// TIA Portal project "漳州" (V17)

(* hardware
DEVICE "S7-1200 station_1"  S7-1200 Station
   slot 0: "Rack_0"  S7-1200 Rack  Rack  V1.0
   slot 1: "PLC_1"  CPU 1215C AC/DC/Rly  6ES7 215-1BG40-0XB0  V4.3
   slot 2: "DI 16x24VDC/DQ 16xRelay_1"  SM 1223 DI16/DQ16 x relay  6ES7 223-1PL32-0XB0  V2.0
*)

// ===== PLC "PLC_1"  CPU 1215C AC/DC/Rly =====

VAR_GLOBAL   // PLC tag table "默认变量表"
   "启动" AT %I0.0 : Bool;
   "停止" AT %I0.1 : Bool;
   "变频器故障" AT %I0.5 : Bool;
   "有料检测" AT %I0.6 : Bool;
   "自动模式" AT %I0.3 : Bool;
   "分拣选择" AT %I0.2 : Bool;
   "变频器运行" AT %Q0.0 : Bool;
   "变频器速段" AT %Q0.1 : Bool;
   "1组正运行" AT %Q2.0 : Bool;
   "Tag_1" AT %Q3.0 : Bool;
   "2组正运行" AT %Q2.2 : Bool;
   "3组正运行" AT %Q2.4 : Bool;
   "4组正运行" AT %Q2.6 : Bool;
   "1组反转(1)" AT %Q2.1 : Bool;
   "2组反转(1)" AT %Q2.3 : Bool;
   "3组反转(1)" AT %Q2.5 : Bool;
   "4组反转(1)" AT %Q2.7 : Bool;
   "三基色绿色" AT %Q0.2 : Bool;
   "三基色红色" AT %Q0.4 : Bool;
   "蜂鸣器" AT %Q0.5 : Bool;
   "Tag_27" AT %Q3.1 : Bool;
   "Tag_28" AT %Q3.3 : Bool;
   "Tag_29" AT %Q3.5 : Bool;
   "Tag_30" AT %Q3.7 : Bool;
   "System_Byte" AT %MB1 : Byte;
   "FirstScan" AT %M1.0 : Bool;
   "DiagStatusUpdate" AT %M1.1 : Bool;
   "AlwaysTRUE" AT %M1.2 : Bool;
   "AlwaysFALSE" AT %M1.3 : Bool;
   "Clock_Byte" AT %MB0 : Byte;
   "Clock_10Hz" AT %M0.0 : Bool;
   "Clock_5Hz" AT %M0.1 : Bool;
   "Clock_2.5Hz" AT %M0.2 : Bool;
   "Clock_2Hz" AT %M0.3 : Bool;
   "Clock_1.25Hz" AT %M0.4 : Bool;
   "Clock_1Hz" AT %M0.5 : Bool;
   "Clock_0.625Hz" AT %M0.6 : Bool;
   "Clock_0.5Hz" AT %M0.7 : Bool;
   "系统启动" AT %M2.0 : Bool;
   "Tag_2" AT %M2.1 : Bool;
   "Tag_3" AT %MW100 : Word;
   "Tag_4" AT %M2.2 : Bool;
   "1组运转" AT %M3.0 : Bool;
   "1组正转" AT %M3.1 : Bool;
   "2组运转" AT %M3.2 : Bool;
   "2组正转" AT %M3.3 : Bool;
   "Tag_5" AT %M20.0 : Bool;
   "3组运转" AT %M3.4 : Bool;
   "3组正转" AT %M3.5 : Bool;
   "4组运转" AT %M3.6 : Bool;
   "4组正转" AT %M3.7 : Bool;
   "1组反运行" AT %M4.0 : Bool;
   "1组反转" AT %M4.1 : Bool;
   "2组反运转" AT %M4.2 : Bool;
   "2组反转" AT %M4.3 : Bool;
   "3组反运行" AT %M4.4 : Bool;
   "3组反转" AT %M4.5 : Bool;
   "4组反运行" AT %M4.6 : Bool;
   "4组反转" AT %M4.7 : Bool;
   "Tag_6" AT %M20.1 : Bool;
   "Tag_7" AT %M20.2 : Bool;
   "Tag_8" AT %M20.3 : Bool;
   "Tag_9" AT %MW200 : Int;
   "Tag_10" AT %MW201 : Int;
   "Tag_11" AT %MW202 : Int;
   "Tag_12" AT %MW203 : Int;
   "Tag_13" AT %MW204 : Int;
   "Tag_14" AT %MW205 : Int;
   "Tag_15" AT %MW206 : Int;
   "Tag_16" AT %MW300 : Int;
   "Tag_17" AT %MW302 : Int;
   "Tag_18" AT %MW304 : Int;
   "Tag_19" AT %MW306 : Int;
   "Tag_20" AT %M110.0 : Bool;
   "Tag_21" AT %MD200 : DWord;
   "Tag_22" AT %MD300 : DWord;
   "Tag_23" AT %MD204 : DWord;
   "Tag_24" AT %MD304 : DWord;
   "Tag_25" AT %M100.0 : Bool;
   "Tag_26" AT %M200.0 : Bool;
   "Tag_31" AT %M200.1 : Bool;
   "Tag_32" AT %M200.2 : Bool;
   "Tag_33" AT %M300.0 : Bool;
   "Tag_34" AT %M5.2 : Bool;
   "Tag_35" AT %M5.3 : Bool;
   "Tag_36" AT %M5.4 : Bool;
   "Tag_37" AT %M11.0 : Bool;
   "Tag_38" AT %M101.0 : Bool;
   "Tag_39" AT %M12.0 : Bool;
   "Tag_40" AT %M12.1 : Bool;
   "Tag_41" AT %M12.2 : Bool;
   "Tag_42" AT %M12.3 : Bool;
   "Tag_43" AT %M12.4 : Bool;
   "Tag_44" AT %M12.5 : Bool;
   "Tag_45" AT %M12.6 : Bool;
   "Tag_46" AT %MB10 : Byte;
   "5组正转" AT %M5.0 : Bool;
   "Tag_48" AT %M6.1 : Bool;
   "Tag_49" AT %M6.2 : Bool;
   "Tag_50" AT %M6.3 : Bool;
   "Tag_51" AT %M6.4 : Bool;
   "Tag_52" AT %M6.5 : Bool;
   "Tag_53" AT %M6.6 : Bool;
   "Tag_54" AT %M6.7 : Bool;
   "Tag_55" AT %M6.0 : Bool;
   "Tag_56" AT %M90.3 : Bool;
   "Tag_57" AT %M90.5 : Bool;
   "Tag_58" AT %M90.0 : Bool;
   "Tag_59" AT %M7.0 : Bool;
   "Tag_60" AT %M7.1 : Bool;
   "Tag_61" AT %M90.2 : Bool;
   "Tag_62" AT %M90.1 : Bool;
   "Tag_63" AT %M7.2 : Bool;
   "Tag_64" AT %M7.3 : Bool;
   "Tag_65" AT %M90.4 : Bool;
   "Tag_66" AT %M7.4 : Bool;
   "Tag_67" AT %M7.5 : Bool;
   "Tag_68" AT %M7.6 : Bool;
   "Tag_69" AT %M8.0 : Bool;
   "Tag_70" AT %M8.1 : Bool;
   "Tag_71" AT %M8.2 : Bool;
   "Tag_72" AT %M8.3 : Bool;
   "Tag_73" AT %M8.4 : Bool;
   "Tag_74" AT %M8.5 : Bool;
   "Tag_75" AT %M8.6 : Bool;
   "Tag_76" AT %M8.7 : Bool;
   "5组反转" AT %M5.1 : Bool;
   "Tag_78" AT %MW102 : Word;
   "Tag_79" AT %MB100 : Byte;
   "Tag_80" AT %M5.5 : Bool;
   "1-1口计时" AT %M10.0 : Bool;
   "1-2计时" AT %M10.1 : Bool;
   "Tag_82" AT %Q10.0 : Bool;
   "Tag_83" AT %M101.1 : Bool;
   "Tag_84" AT %M101.2 : Bool;
   "Tag_81" AT %Q10.1 : Bool;
   "Tag_85" AT %M101.3 : Bool;
   "Tag_86" AT %M10.2 : Bool;
   "Tag_87" AT %Q10.2 : Bool;
   "Tag_88" AT %M101.4 : Bool;
   "Tag_89" AT %M10.3 : Bool;
   "Tag_90" AT %M101.5 : Bool;
   "Tag_91" AT %M101.6 : Bool;
   "Tag_92" AT %M101.7 : Bool;
   "Tag_93" AT %MB101 : Byte;
   "Tag_94" AT %M100.1 : Bool;
   "Tag_95" AT %M100.2 : Bool;
   "Tag_96" AT %M100.3 : Bool;
   "Tag_97" AT %M100.4 : Bool;
   "Tag_98" AT %MB102 : Byte;
   "Tag_99" AT %MB103 : Byte;
   "Tag_100" AT %M103.1 : Bool;
   "Tag_101" AT %M102.2 : Bool;
   "Tag_102" AT %M102.3 : Bool;
   "Tag_103" AT %M102.4 : Bool;
   "Tag_104" AT %M103.2 : Bool;
   "Tag_105" AT %M103.3 : Bool;
   "Tag_106" AT %M103.4 : Bool;
   "Tag_107" AT %M102.1 : Bool;
   "Tag_108" AT %MB104 : Byte;
   "Tag_109" AT %MB105 : Byte;
   "Tag_110" AT %M105.1 : Bool;
   "Tag_111" AT %M105.2 : Bool;
   "Tag_112" AT %M105.3 : Bool;
   "Tag_113" AT %M105.4 : Bool;
   "Tag_114" AT %M104.1 : Bool;
   "Tag_115" AT %M104.2 : Bool;
   "Tag_116" AT %M104.3 : Bool;
   "Tag_117" AT %MB106 : Byte;
   "Tag_118" AT %MB107 : Byte;
   "Tag_119" AT %M107.1 : Bool;
   "Tag_120" AT %M107.2 : Bool;
   "Tag_121" AT %M107.3 : Bool;
   "Tag_122" AT %M107.4 : Bool;
   "Tag_123" AT %M106.1 : Bool;
   "Tag_124" AT %M106.2 : Bool;
   "Tag_125" AT %M106.3 : Bool;
   "Tag_126" AT %M106.4 : Bool;
   "Tag_127" AT %MB108 : Byte;
   "Tag_128" AT %MB109 : Byte;
   "Tag_129" AT %M109.1 : Bool;
   "Tag_130" AT %M109.2 : Bool;
   "Tag_131" AT %M109.3 : Bool;
   "Tag_132" AT %M109.4 : Bool;
   "Tag_133" AT %M109.5 : Bool;
   "Tag_134" AT %M108.1 : Bool;
   "Tag_135" AT %M108.2 : Bool;
   "Tag_136" AT %M108.3 : Bool;
   "Tag_137" AT %M108.4 : Bool;
   "Tag_138" AT %M108.5 : Bool;
END_VAR

TYPE "用户数据类型_1"
   STRUCT
      Q : Array[0..12] of Bool;
   END_STRUCT;
END_TYPE

DATA_BLOCK "1口_DB"   // DB1
{ S7_Optimized_Access := 'TRUE' }
VERSION : 0.1
// stored: InstanceOfName 1口
"1口"
BEGIN
END_DATA_BLOCK

DATA_BLOCK "2口_DB"   // DB2
{ S7_Optimized_Access := 'TRUE' }
VERSION : 0.1
// stored: InstanceOfName 2口
"2口"
BEGIN
END_DATA_BLOCK

DATA_BLOCK "3口_DB"   // DB3
{ S7_Optimized_Access := 'TRUE' }
VERSION : 0.1
// stored: InstanceOfName 3口
"3口"
BEGIN
END_DATA_BLOCK

DATA_BLOCK "4口_DB"   // DB4
{ S7_Optimized_Access := 'TRUE' }
VERSION : 0.1
// stored: InstanceOfName 4口
"4口"
BEGIN
END_DATA_BLOCK

DATA_BLOCK "数据块_1"   // DB5
{ S7_Optimized_Access := 'TRUE' }
VERSION : 0.1
   VAR
      箱号 : Int;
      分拣时间 : Time := T#1s;
      到达时间 : Time := T#10s;
      光电 : Bool;
      计数 : Bool;
      Q : Array[0..12] of Bool;
   END_VAR
BEGIN
END_DATA_BLOCK

DATA_BLOCK "5口_DB"   // DB6
{ S7_Optimized_Access := 'TRUE' }
VERSION : 0.1
// stored: InstanceOfName 5口
"5口"
BEGIN
END_DATA_BLOCK

FUNCTION_BLOCK "1口"   // FB1, LAD
{ S7_Optimized_Access := 'TRUE' }
VERSION : 0.1
   VAR_INPUT
      光电 : Bool;
      箱号 : Int;
   END_VAR
   VAR_OUTPUT
      Q : Array[0..12] of Bool;
   END_VAR
   VAR
      TON_TIME : Array[0..21] of TON_TIME;
      IEC_Timer : Array[0..11] of IEC_TIMER;
      "M" : Array[0..11] of Bool;
      M1 : Array[0..11] of Bool;
      光电上升沿 : Array[0..2] of Bool;
   END_VAR
   VAR_TEMP   // added for the SCL form of the ladder/FBD networks
      _w1 : Bool;
      _w2 : Bool;
      _w3 : Bool;
   END_VAR
BEGIN

REGION Network 1: 记录箱号
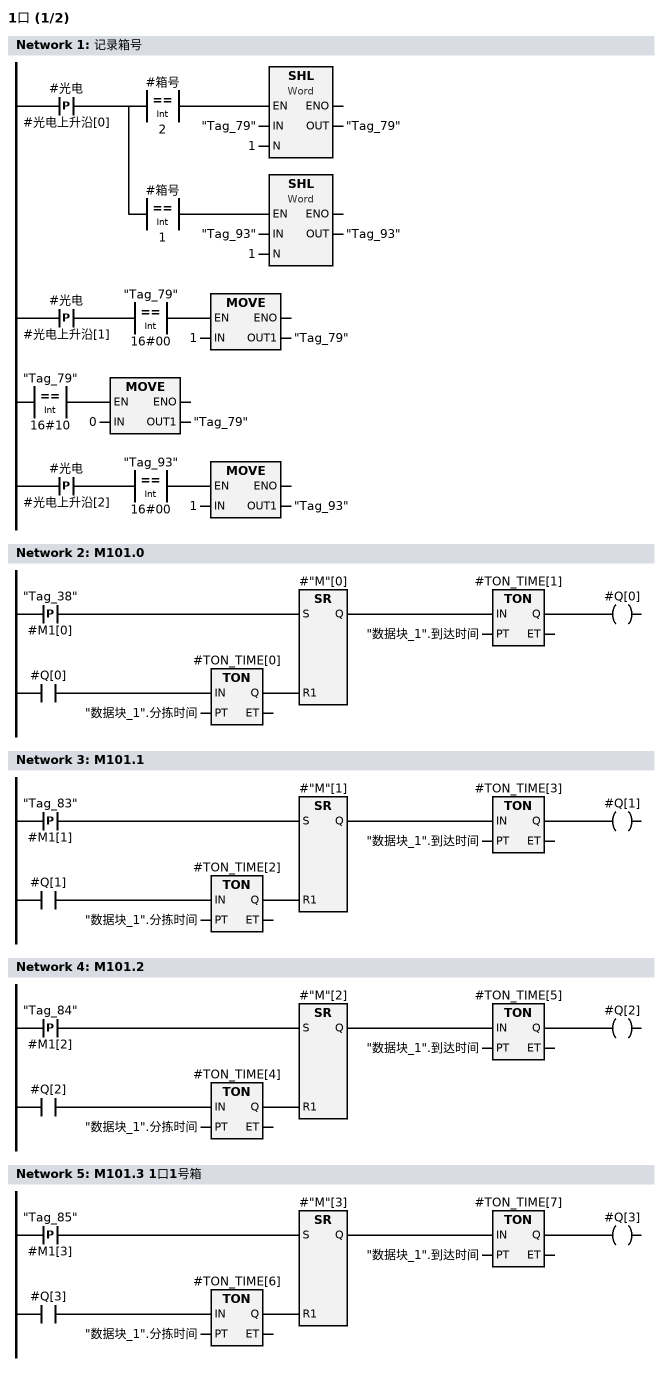
   RUNG wire#powerrail
      P_Contact(operand := #光电, bit := #光电上升沿[0])
      wire#w1
      { S7_Templates := "SrcType := Int" } EQ_Contact(in1 := #箱号, in2 := 2)
      { S7_Templates := "SrcType := Word" } Shl(in := "Tag_79", n := 1, out => "Tag_79")
   END_RUNG
   RUNG wire#w1
      { S7_Templates := "SrcType := Int" } EQ_Contact(in1 := #箱号, in2 := 1)
      { S7_Templates := "SrcType := Word" } Shl(in := "Tag_93", n := 1, out => "Tag_93")
   END_RUNG
   RUNG wire#powerrail
      P_Contact(operand := #光电, bit := #光电上升沿[1])
      { S7_Templates := "SrcType := Int" } EQ_Contact(in1 := "Tag_79", in2 := 16#00)
      Move(in := 1, out1 => "Tag_79")
   END_RUNG
   RUNG wire#powerrail
      { S7_Templates := "SrcType := Int" } EQ_Contact(in1 := "Tag_79", in2 := 16#10)
      Move(in := 0, out1 => "Tag_79")
   END_RUNG
   RUNG wire#powerrail
      P_Contact(operand := #光电, bit := #光电上升沿[2])
      { S7_Templates := "SrcType := Int" } EQ_Contact(in1 := "Tag_93", in2 := 16#00)
      Move(in := 1, out1 => "Tag_93")
   END_RUNG
   // the same network as SCL:
   #_w1 := #光电 AND NOT #光电上升沿[0];   // rising edge of #光电
   #光电上升沿[0] := #光电;
   IF #_w1 AND (#箱号 = 2) THEN "Tag_79" := SHL(IN := "Tag_79", N := 1); END_IF;
   IF #_w1 AND (#箱号 = 1) THEN "Tag_93" := SHL(IN := "Tag_93", N := 1); END_IF;
   #_w2 := #光电 AND NOT #光电上升沿[1];   // rising edge of #光电
   #光电上升沿[1] := #光电;
   IF #_w2 AND ("Tag_79" = 16#00) THEN "Tag_79" := 1; END_IF;
   IF "Tag_79" = 16#10 THEN "Tag_79" := 0; END_IF;
   #_w3 := #光电 AND NOT #光电上升沿[2];   // rising edge of #光电
   #光电上升沿[2] := #光电;
   IF #_w3 AND ("Tag_93" = 16#00) THEN "Tag_93" := 1; END_IF;
END_REGION

REGION Network 2: M101.0
   #_w1 := "Tag_38" AND NOT #M1[0];   // rising edge of "Tag_38"
   #M1[0] := "Tag_38";
   #TON_TIME[0].TON(IN := #Q[0], PT := "数据块_1".分拣时间);
   IF #_w1 THEN
       #"M"[0] := TRUE;   // SR flip-flop
   END_IF;
   IF #TON_TIME[0].Q THEN #"M"[0] := FALSE; END_IF;
   #TON_TIME[1].TON(IN := #"M"[0], PT := "数据块_1".到达时间);
   #Q[0] := #TON_TIME[1].Q;
END_REGION

REGION Network 3: M101.1
   #_w1 := "Tag_83" AND NOT #M1[1];   // rising edge of "Tag_83"
   #M1[1] := "Tag_83";
   #TON_TIME[2].TON(IN := #Q[1], PT := "数据块_1".分拣时间);
   IF #_w1 THEN
       #"M"[1] := TRUE;   // SR flip-flop
   END_IF;
   IF #TON_TIME[2].Q THEN #"M"[1] := FALSE; END_IF;
   #TON_TIME[3].TON(IN := #"M"[1], PT := "数据块_1".到达时间);
   #Q[1] := #TON_TIME[3].Q;
END_REGION

REGION Network 4: M101.2
   #_w1 := "Tag_84" AND NOT #M1[2];   // rising edge of "Tag_84"
   #M1[2] := "Tag_84";
   #TON_TIME[4].TON(IN := #Q[2], PT := "数据块_1".分拣时间);
   IF #_w1 THEN
       #"M"[2] := TRUE;   // SR flip-flop
   END_IF;
   IF #TON_TIME[4].Q THEN #"M"[2] := FALSE; END_IF;
   #TON_TIME[5].TON(IN := #"M"[2], PT := "数据块_1".到达时间);
   #Q[2] := #TON_TIME[5].Q;
END_REGION

REGION Network 5: M101.3 1口1号箱
   #_w1 := "Tag_85" AND NOT #M1[3];   // rising edge of "Tag_85"
   #M1[3] := "Tag_85";
   #TON_TIME[6].TON(IN := #Q[3], PT := "数据块_1".分拣时间);
   IF #_w1 THEN
       #"M"[3] := TRUE;   // SR flip-flop
   END_IF;
   IF #TON_TIME[6].Q THEN #"M"[3] := FALSE; END_IF;
   #TON_TIME[7].TON(IN := #"M"[3], PT := "数据块_1".到达时间);
   #Q[3] := #TON_TIME[7].Q;
END_REGION

REGION Network 6: M100.0 1口2号箱
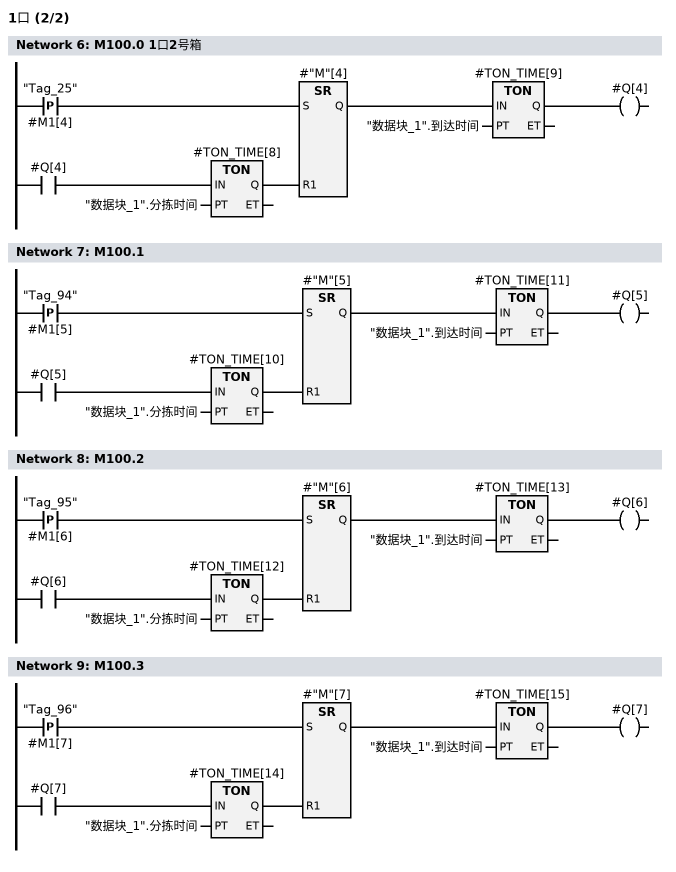
   #_w1 := "Tag_25" AND NOT #M1[4];   // rising edge of "Tag_25"
   #M1[4] := "Tag_25";
   #TON_TIME[8].TON(IN := #Q[4], PT := "数据块_1".分拣时间);
   IF #_w1 THEN
       #"M"[4] := TRUE;   // SR flip-flop
   END_IF;
   IF #TON_TIME[8].Q THEN #"M"[4] := FALSE; END_IF;
   #TON_TIME[9].TON(IN := #"M"[4], PT := "数据块_1".到达时间);
   #Q[4] := #TON_TIME[9].Q;
END_REGION

REGION Network 7: M100.1
   #_w1 := "Tag_94" AND NOT #M1[5];   // rising edge of "Tag_94"
   #M1[5] := "Tag_94";
   #TON_TIME[10].TON(IN := #Q[5], PT := "数据块_1".分拣时间);
   IF #_w1 THEN
       #"M"[5] := TRUE;   // SR flip-flop
   END_IF;
   IF #TON_TIME[10].Q THEN #"M"[5] := FALSE; END_IF;
   #TON_TIME[11].TON(IN := #"M"[5], PT := "数据块_1".到达时间);
   #Q[5] := #TON_TIME[11].Q;
END_REGION

REGION Network 8: M100.2
   #_w1 := "Tag_95" AND NOT #M1[6];   // rising edge of "Tag_95"
   #M1[6] := "Tag_95";
   #TON_TIME[12].TON(IN := #Q[6], PT := "数据块_1".分拣时间);
   IF #_w1 THEN
       #"M"[6] := TRUE;   // SR flip-flop
   END_IF;
   IF #TON_TIME[12].Q THEN #"M"[6] := FALSE; END_IF;
   #TON_TIME[13].TON(IN := #"M"[6], PT := "数据块_1".到达时间);
   #Q[6] := #TON_TIME[13].Q;
END_REGION

REGION Network 9: M100.3
   #_w1 := "Tag_96" AND NOT #M1[7];   // rising edge of "Tag_96"
   #M1[7] := "Tag_96";
   #TON_TIME[14].TON(IN := #Q[7], PT := "数据块_1".分拣时间);
   IF #_w1 THEN
       #"M"[7] := TRUE;   // SR flip-flop
   END_IF;
   IF #TON_TIME[14].Q THEN #"M"[7] := FALSE; END_IF;
   #TON_TIME[15].TON(IN := #"M"[7], PT := "数据块_1".到达时间);
   #Q[7] := #TON_TIME[15].Q;
END_REGION

REGION Network 10 (SCL)
   IF #Q[0] OR #Q[1] OR #Q[2] OR #Q[3] THEN
       "1组正转" := TRUE;
   ELSE
       "1组正转" := FALSE;
   END_IF;

   IF #Q[4] OR #Q[5] OR #Q[6] OR #Q[7] THEN
       "1组反转" := TRUE;
   ELSE
       "1组反转" := FALSE;
   END_IF;
END_REGION
END_FUNCTION_BLOCK

FUNCTION_BLOCK "2口"   // FB2, LAD
{ S7_Optimized_Access := 'TRUE' }
VERSION : 0.1
   VAR_INPUT
      光电 : Bool;
      箱号 : Int;
   END_VAR
   VAR_OUTPUT
      Q : Array[0..12] of Bool;
   END_VAR
   VAR
      TON_TIME : Array[0..21] of TON_TIME;
      IEC_Timer : Array[0..11] of IEC_TIMER;
      "M" : Array[0..11] of Bool;
      M1 : Array[0..11] of Bool;
      光电上升沿 : Bool;
   END_VAR
   VAR_TEMP   // added for the SCL form of the ladder/FBD networks
      _w1 : Bool;
      _w2 : Bool;
      _w3 : Bool;
   END_VAR
BEGIN

REGION Network 1: 记录箱号
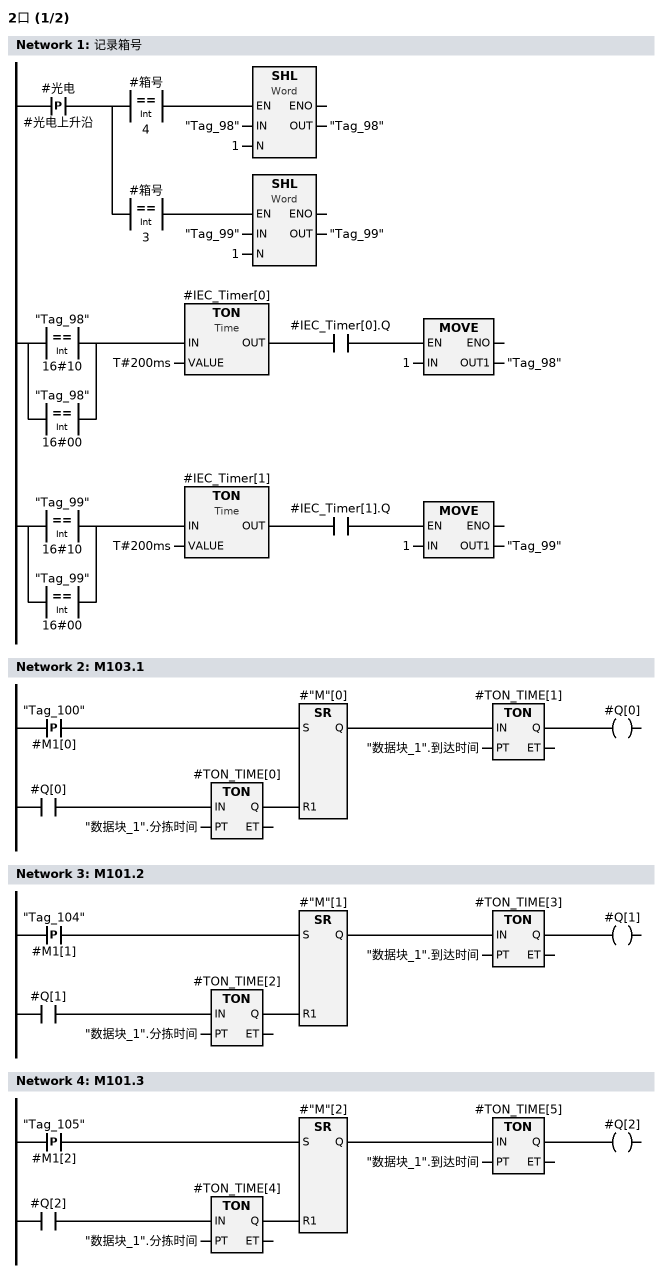
   #_w1 := #光电 AND NOT #光电上升沿;   // rising edge of #光电
   #光电上升沿 := #光电;
   IF #_w1 AND (#箱号 = 4) THEN "Tag_98" := SHL(IN := "Tag_98", N := 1); END_IF;
   IF #_w1 AND (#箱号 = 3) THEN "Tag_99" := SHL(IN := "Tag_99", N := 1); END_IF;
   #_w2 := ("Tag_98" = 16#10) OR ("Tag_98" = 16#00);
   #IEC_Timer[0].TON(IN := #_w2, PT := T#200ms);   // TON coil
   IF #_w2 AND #IEC_Timer[0].Q THEN "Tag_98" := 1; END_IF;
   #_w3 := ("Tag_99" = 16#10) OR ("Tag_99" = 16#00);
   #IEC_Timer[1].TON(IN := #_w3, PT := T#200ms);   // TON coil
   IF #_w3 AND #IEC_Timer[1].Q THEN "Tag_99" := 1; END_IF;
END_REGION

REGION Network 2: M103.1
   #_w1 := "Tag_100" AND NOT #M1[0];   // rising edge of "Tag_100"
   #M1[0] := "Tag_100";
   #TON_TIME[0].TON(IN := #Q[0], PT := "数据块_1".分拣时间);
   IF #_w1 THEN
       #"M"[0] := TRUE;   // SR flip-flop
   END_IF;
   IF #TON_TIME[0].Q THEN #"M"[0] := FALSE; END_IF;
   #TON_TIME[1].TON(IN := #"M"[0], PT := "数据块_1".到达时间);
   #Q[0] := #TON_TIME[1].Q;
END_REGION

REGION Network 3: M101.2
   #_w1 := "Tag_104" AND NOT #M1[1];   // rising edge of "Tag_104"
   #M1[1] := "Tag_104";
   #TON_TIME[2].TON(IN := #Q[1], PT := "数据块_1".分拣时间);
   IF #_w1 THEN
       #"M"[1] := TRUE;   // SR flip-flop
   END_IF;
   IF #TON_TIME[2].Q THEN #"M"[1] := FALSE; END_IF;
   #TON_TIME[3].TON(IN := #"M"[1], PT := "数据块_1".到达时间);
   #Q[1] := #TON_TIME[3].Q;
END_REGION

REGION Network 4: M101.3
   #_w1 := "Tag_105" AND NOT #M1[2];   // rising edge of "Tag_105"
   #M1[2] := "Tag_105";
   #TON_TIME[4].TON(IN := #Q[2], PT := "数据块_1".分拣时间);
   IF #_w1 THEN
       #"M"[2] := TRUE;   // SR flip-flop
   END_IF;
   IF #TON_TIME[4].Q THEN #"M"[2] := FALSE; END_IF;
   #TON_TIME[5].TON(IN := #"M"[2], PT := "数据块_1".到达时间);
   #Q[2] := #TON_TIME[5].Q;
END_REGION

REGION Network 5: M101.4 1口1号箱
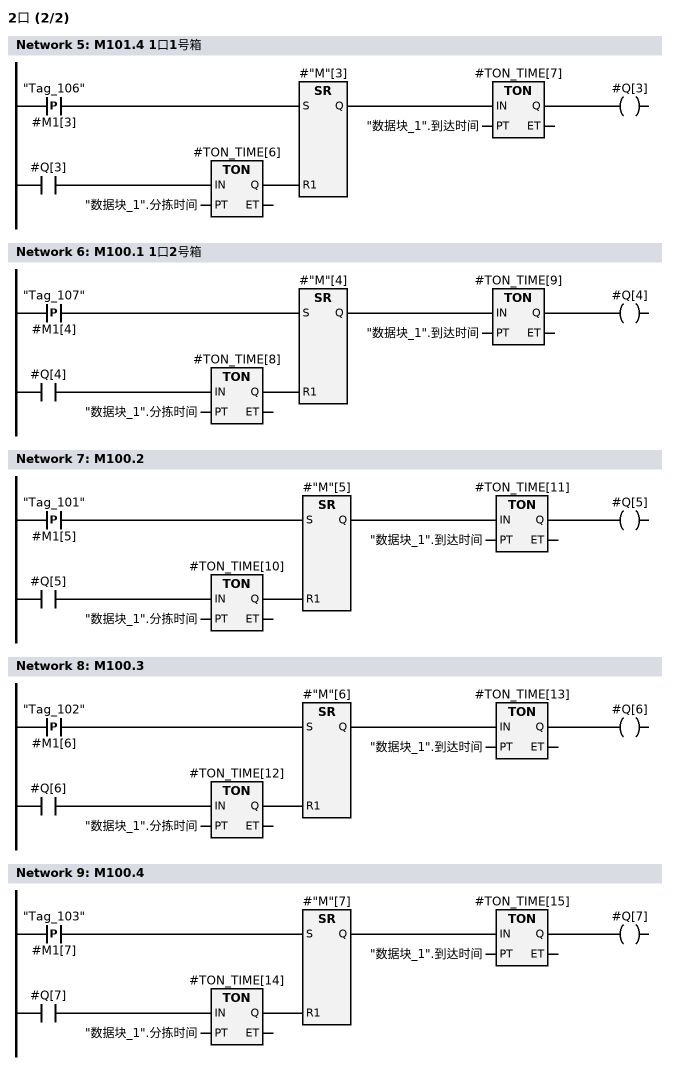
   #_w1 := "Tag_106" AND NOT #M1[3];   // rising edge of "Tag_106"
   #M1[3] := "Tag_106";
   #TON_TIME[6].TON(IN := #Q[3], PT := "数据块_1".分拣时间);
   IF #_w1 THEN
       #"M"[3] := TRUE;   // SR flip-flop
   END_IF;
   IF #TON_TIME[6].Q THEN #"M"[3] := FALSE; END_IF;
   #TON_TIME[7].TON(IN := #"M"[3], PT := "数据块_1".到达时间);
   #Q[3] := #TON_TIME[7].Q;
END_REGION

REGION Network 6: M100.1 1口2号箱
   #_w1 := "Tag_107" AND NOT #M1[4];   // rising edge of "Tag_107"
   #M1[4] := "Tag_107";
   #TON_TIME[8].TON(IN := #Q[4], PT := "数据块_1".分拣时间);
   IF #_w1 THEN
       #"M"[4] := TRUE;   // SR flip-flop
   END_IF;
   IF #TON_TIME[8].Q THEN #"M"[4] := FALSE; END_IF;
   #TON_TIME[9].TON(IN := #"M"[4], PT := "数据块_1".到达时间);
   #Q[4] := #TON_TIME[9].Q;
END_REGION

REGION Network 7: M100.2
   #_w1 := "Tag_101" AND NOT #M1[5];   // rising edge of "Tag_101"
   #M1[5] := "Tag_101";
   #TON_TIME[10].TON(IN := #Q[5], PT := "数据块_1".分拣时间);
   IF #_w1 THEN
       #"M"[5] := TRUE;   // SR flip-flop
   END_IF;
   IF #TON_TIME[10].Q THEN #"M"[5] := FALSE; END_IF;
   #TON_TIME[11].TON(IN := #"M"[5], PT := "数据块_1".到达时间);
   #Q[5] := #TON_TIME[11].Q;
END_REGION

REGION Network 8: M100.3
   #_w1 := "Tag_102" AND NOT #M1[6];   // rising edge of "Tag_102"
   #M1[6] := "Tag_102";
   #TON_TIME[12].TON(IN := #Q[6], PT := "数据块_1".分拣时间);
   IF #_w1 THEN
       #"M"[6] := TRUE;   // SR flip-flop
   END_IF;
   IF #TON_TIME[12].Q THEN #"M"[6] := FALSE; END_IF;
   #TON_TIME[13].TON(IN := #"M"[6], PT := "数据块_1".到达时间);
   #Q[6] := #TON_TIME[13].Q;
END_REGION

REGION Network 9: M100.4
   #_w1 := "Tag_103" AND NOT #M1[7];   // rising edge of "Tag_103"
   #M1[7] := "Tag_103";
   #TON_TIME[14].TON(IN := #Q[7], PT := "数据块_1".分拣时间);
   IF #_w1 THEN
       #"M"[7] := TRUE;   // SR flip-flop
   END_IF;
   IF #TON_TIME[14].Q THEN #"M"[7] := FALSE; END_IF;
   #TON_TIME[15].TON(IN := #"M"[7], PT := "数据块_1".到达时间);
   #Q[7] := #TON_TIME[15].Q;
END_REGION

REGION Network 10 (SCL)
   IF #Q[0] OR #Q[1] OR #Q[2] OR #Q[3] THEN
       "2组正转" := TRUE;
   ELSE
       "2组正转" := FALSE;
   END_IF;

   IF #Q[4] OR #Q[5] OR #Q[6] OR #Q[7] THEN
       "2组反转" := TRUE;
   ELSE
       "2组反转" := FALSE;
   END_IF;
END_REGION
END_FUNCTION_BLOCK

FUNCTION_BLOCK "3口"   // FB3, LAD
{ S7_Optimized_Access := 'TRUE' }
VERSION : 0.1
   VAR_INPUT
      光电 : Bool;
      箱号 : Int;
   END_VAR
   VAR_OUTPUT
      Q : Array[0..12] of Bool;
   END_VAR
   VAR
      TON_TIME : Array[0..21] of TON_TIME;
      IEC_Timer : Array[0..11] of IEC_TIMER;
      "M" : Array[0..11] of Bool;
      M1 : Array[0..11] of Bool;
      光电上升沿 : Bool;
   END_VAR
   VAR_TEMP   // added for the SCL form of the ladder/FBD networks
      _w1 : Bool;
      _w2 : Bool;
      _w3 : Bool;
   END_VAR
BEGIN

REGION Network 1: 记录箱号
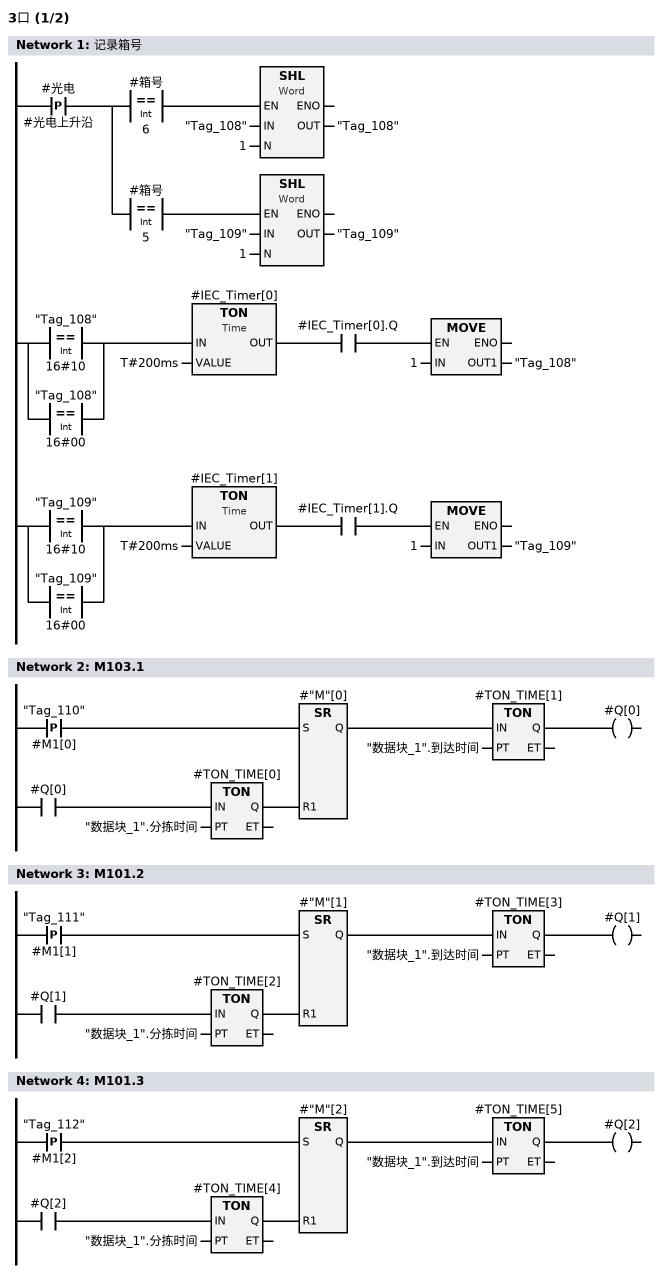
   #_w1 := #光电 AND NOT #光电上升沿;   // rising edge of #光电
   #光电上升沿 := #光电;
   IF #_w1 AND (#箱号 = 6) THEN "Tag_108" := SHL(IN := "Tag_108", N := 1); END_IF;
   IF #_w1 AND (#箱号 = 5) THEN "Tag_109" := SHL(IN := "Tag_109", N := 1); END_IF;
   #_w2 := ("Tag_108" = 16#10) OR ("Tag_108" = 16#00);
   #IEC_Timer[0].TON(IN := #_w2, PT := T#200ms);   // TON coil
   IF #_w2 AND #IEC_Timer[0].Q THEN "Tag_108" := 1; END_IF;
   #_w3 := ("Tag_109" = 16#10) OR ("Tag_109" = 16#00);
   #IEC_Timer[1].TON(IN := #_w3, PT := T#200ms);   // TON coil
   IF #_w3 AND #IEC_Timer[1].Q THEN "Tag_109" := 1; END_IF;
END_REGION

REGION Network 2: M103.1
   #_w1 := "Tag_110" AND NOT #M1[0];   // rising edge of "Tag_110"
   #M1[0] := "Tag_110";
   #TON_TIME[0].TON(IN := #Q[0], PT := "数据块_1".分拣时间);
   IF #_w1 THEN
       #"M"[0] := TRUE;   // SR flip-flop
   END_IF;
   IF #TON_TIME[0].Q THEN #"M"[0] := FALSE; END_IF;
   #TON_TIME[1].TON(IN := #"M"[0], PT := "数据块_1".到达时间);
   #Q[0] := #TON_TIME[1].Q;
END_REGION

REGION Network 3: M101.2
   #_w1 := "Tag_111" AND NOT #M1[1];   // rising edge of "Tag_111"
   #M1[1] := "Tag_111";
   #TON_TIME[2].TON(IN := #Q[1], PT := "数据块_1".分拣时间);
   IF #_w1 THEN
       #"M"[1] := TRUE;   // SR flip-flop
   END_IF;
   IF #TON_TIME[2].Q THEN #"M"[1] := FALSE; END_IF;
   #TON_TIME[3].TON(IN := #"M"[1], PT := "数据块_1".到达时间);
   #Q[1] := #TON_TIME[3].Q;
END_REGION

REGION Network 4: M101.3
   #_w1 := "Tag_112" AND NOT #M1[2];   // rising edge of "Tag_112"
   #M1[2] := "Tag_112";
   #TON_TIME[4].TON(IN := #Q[2], PT := "数据块_1".分拣时间);
   IF #_w1 THEN
       #"M"[2] := TRUE;   // SR flip-flop
   END_IF;
   IF #TON_TIME[4].Q THEN #"M"[2] := FALSE; END_IF;
   #TON_TIME[5].TON(IN := #"M"[2], PT := "数据块_1".到达时间);
   #Q[2] := #TON_TIME[5].Q;
END_REGION

REGION Network 5: M101.4 1口1号箱
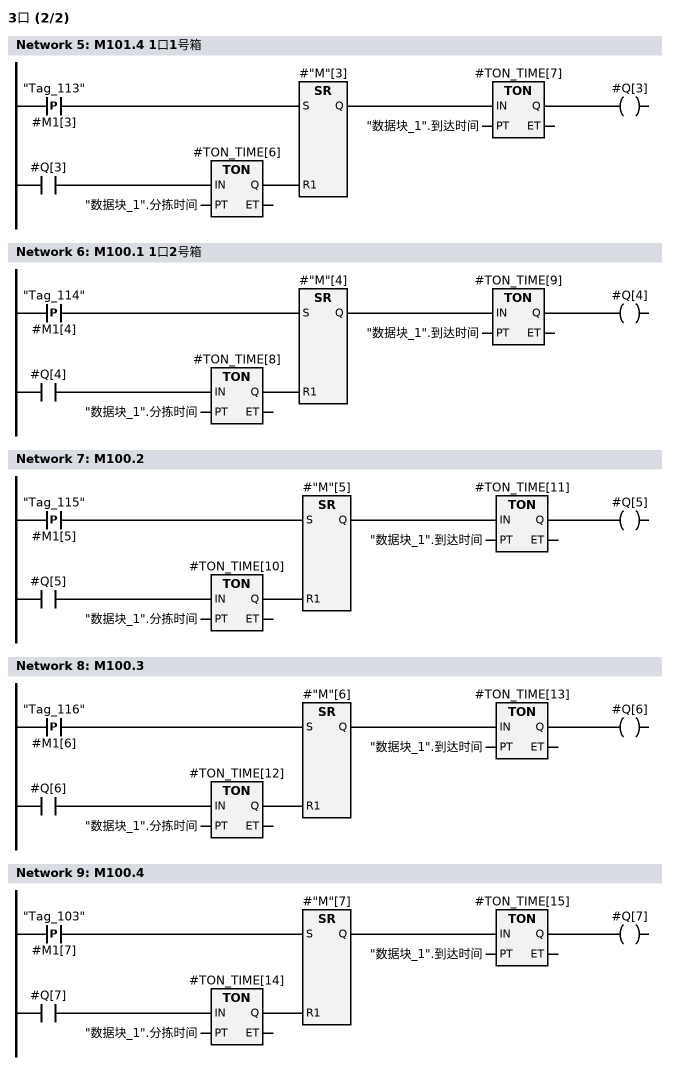
   #_w1 := "Tag_113" AND NOT #M1[3];   // rising edge of "Tag_113"
   #M1[3] := "Tag_113";
   #TON_TIME[6].TON(IN := #Q[3], PT := "数据块_1".分拣时间);
   IF #_w1 THEN
       #"M"[3] := TRUE;   // SR flip-flop
   END_IF;
   IF #TON_TIME[6].Q THEN #"M"[3] := FALSE; END_IF;
   #TON_TIME[7].TON(IN := #"M"[3], PT := "数据块_1".到达时间);
   #Q[3] := #TON_TIME[7].Q;
END_REGION

REGION Network 6: M100.1 1口2号箱
   #_w1 := "Tag_114" AND NOT #M1[4];   // rising edge of "Tag_114"
   #M1[4] := "Tag_114";
   #TON_TIME[8].TON(IN := #Q[4], PT := "数据块_1".分拣时间);
   IF #_w1 THEN
       #"M"[4] := TRUE;   // SR flip-flop
   END_IF;
   IF #TON_TIME[8].Q THEN #"M"[4] := FALSE; END_IF;
   #TON_TIME[9].TON(IN := #"M"[4], PT := "数据块_1".到达时间);
   #Q[4] := #TON_TIME[9].Q;
END_REGION

REGION Network 7: M100.2
   #_w1 := "Tag_115" AND NOT #M1[5];   // rising edge of "Tag_115"
   #M1[5] := "Tag_115";
   #TON_TIME[10].TON(IN := #Q[5], PT := "数据块_1".分拣时间);
   IF #_w1 THEN
       #"M"[5] := TRUE;   // SR flip-flop
   END_IF;
   IF #TON_TIME[10].Q THEN #"M"[5] := FALSE; END_IF;
   #TON_TIME[11].TON(IN := #"M"[5], PT := "数据块_1".到达时间);
   #Q[5] := #TON_TIME[11].Q;
END_REGION

REGION Network 8: M100.3
   #_w1 := "Tag_116" AND NOT #M1[6];   // rising edge of "Tag_116"
   #M1[6] := "Tag_116";
   #TON_TIME[12].TON(IN := #Q[6], PT := "数据块_1".分拣时间);
   IF #_w1 THEN
       #"M"[6] := TRUE;   // SR flip-flop
   END_IF;
   IF #TON_TIME[12].Q THEN #"M"[6] := FALSE; END_IF;
   #TON_TIME[13].TON(IN := #"M"[6], PT := "数据块_1".到达时间);
   #Q[6] := #TON_TIME[13].Q;
END_REGION

REGION Network 9: M100.4
   #_w1 := "Tag_103" AND NOT #M1[7];   // rising edge of "Tag_103"
   #M1[7] := "Tag_103";
   #TON_TIME[14].TON(IN := #Q[7], PT := "数据块_1".分拣时间);
   IF #_w1 THEN
       #"M"[7] := TRUE;   // SR flip-flop
   END_IF;
   IF #TON_TIME[14].Q THEN #"M"[7] := FALSE; END_IF;
   #TON_TIME[15].TON(IN := #"M"[7], PT := "数据块_1".到达时间);
   #Q[7] := #TON_TIME[15].Q;
END_REGION

REGION Network 10 (SCL)
   REGION 3口6号
       // Statement section REGION
       IF #Q[0] OR #Q[1] OR #Q[2] OR #Q[3] THEN
           "3组正转" := TRUE;
       ELSE
           "3组正转" := FALSE;
       END_IF;
   END_REGION


   REGION 3口5号
       // Statement section REGION
       IF #Q[4] OR #Q[5] OR #Q[6] OR #Q[7] THEN
           "3组反转" := TRUE;
       ELSE
           "3组反转" := FALSE;
       END_IF;
   END_REGION
END_REGION
END_FUNCTION_BLOCK

FUNCTION_BLOCK "4口"   // FB4, LAD
{ S7_Optimized_Access := 'TRUE' }
VERSION : 0.1
   VAR_INPUT
      光电 : Bool;
      箱号 : Int;
   END_VAR
   VAR_OUTPUT
      Q : Array[0..12] of Bool;
   END_VAR
   VAR
      TON_TIME : Array[0..21] of TON_TIME;
      IEC_Timer : Array[0..11] of IEC_TIMER;
      "M" : Array[0..11] of Bool;
      M1 : Array[0..11] of Bool;
      光电上升沿 : Bool;
   END_VAR
   VAR_TEMP   // added for the SCL form of the ladder/FBD networks
      _w1 : Bool;
      _w2 : Bool;
      _w3 : Bool;
   END_VAR
BEGIN

REGION Network 1: 记录箱号
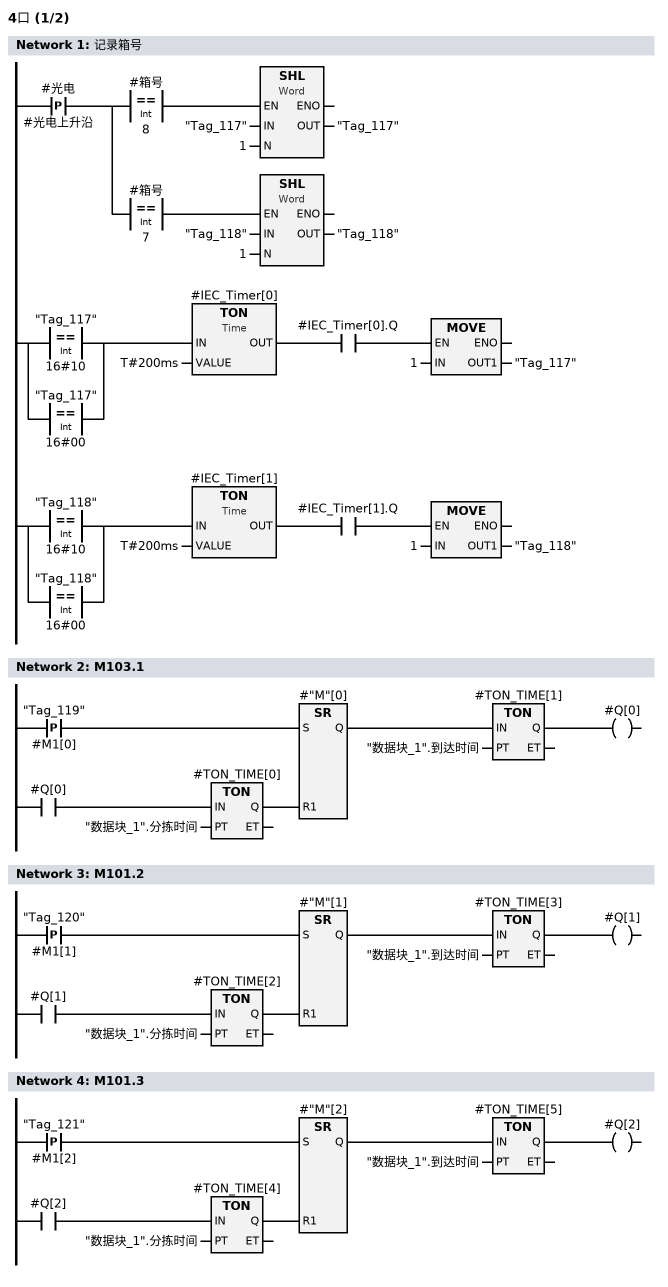
   #_w1 := #光电 AND NOT #光电上升沿;   // rising edge of #光电
   #光电上升沿 := #光电;
   IF #_w1 AND (#箱号 = 8) THEN "Tag_117" := SHL(IN := "Tag_117", N := 1); END_IF;
   IF #_w1 AND (#箱号 = 7) THEN "Tag_118" := SHL(IN := "Tag_118", N := 1); END_IF;
   #_w2 := ("Tag_117" = 16#10) OR ("Tag_117" = 16#00);
   #IEC_Timer[0].TON(IN := #_w2, PT := T#200ms);   // TON coil
   IF #_w2 AND #IEC_Timer[0].Q THEN "Tag_117" := 1; END_IF;
   #_w3 := ("Tag_118" = 16#10) OR ("Tag_118" = 16#00);
   #IEC_Timer[1].TON(IN := #_w3, PT := T#200ms);   // TON coil
   IF #_w3 AND #IEC_Timer[1].Q THEN "Tag_118" := 1; END_IF;
END_REGION

REGION Network 2: M103.1
   #_w1 := "Tag_119" AND NOT #M1[0];   // rising edge of "Tag_119"
   #M1[0] := "Tag_119";
   #TON_TIME[0].TON(IN := #Q[0], PT := "数据块_1".分拣时间);
   IF #_w1 THEN
       #"M"[0] := TRUE;   // SR flip-flop
   END_IF;
   IF #TON_TIME[0].Q THEN #"M"[0] := FALSE; END_IF;
   #TON_TIME[1].TON(IN := #"M"[0], PT := "数据块_1".到达时间);
   #Q[0] := #TON_TIME[1].Q;
END_REGION

REGION Network 3: M101.2
   #_w1 := "Tag_120" AND NOT #M1[1];   // rising edge of "Tag_120"
   #M1[1] := "Tag_120";
   #TON_TIME[2].TON(IN := #Q[1], PT := "数据块_1".分拣时间);
   IF #_w1 THEN
       #"M"[1] := TRUE;   // SR flip-flop
   END_IF;
   IF #TON_TIME[2].Q THEN #"M"[1] := FALSE; END_IF;
   #TON_TIME[3].TON(IN := #"M"[1], PT := "数据块_1".到达时间);
   #Q[1] := #TON_TIME[3].Q;
END_REGION

REGION Network 4: M101.3
   #_w1 := "Tag_121" AND NOT #M1[2];   // rising edge of "Tag_121"
   #M1[2] := "Tag_121";
   #TON_TIME[4].TON(IN := #Q[2], PT := "数据块_1".分拣时间);
   IF #_w1 THEN
       #"M"[2] := TRUE;   // SR flip-flop
   END_IF;
   IF #TON_TIME[4].Q THEN #"M"[2] := FALSE; END_IF;
   #TON_TIME[5].TON(IN := #"M"[2], PT := "数据块_1".到达时间);
   #Q[2] := #TON_TIME[5].Q;
END_REGION

REGION Network 5: M101.4 1口1号箱
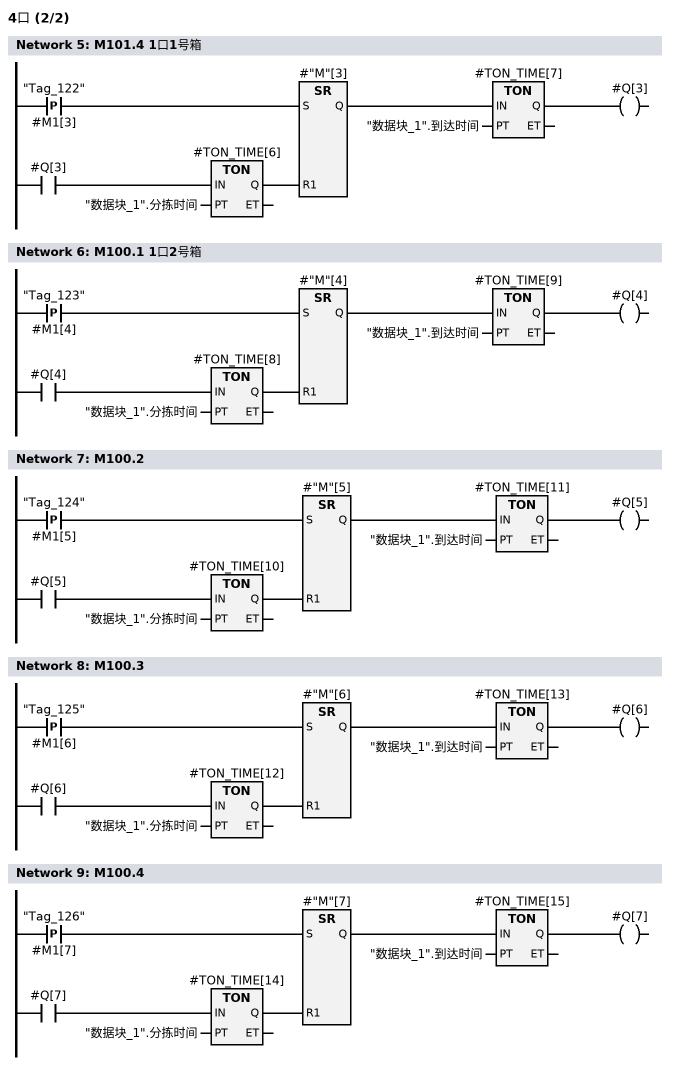
   #_w1 := "Tag_122" AND NOT #M1[3];   // rising edge of "Tag_122"
   #M1[3] := "Tag_122";
   #TON_TIME[6].TON(IN := #Q[3], PT := "数据块_1".分拣时间);
   IF #_w1 THEN
       #"M"[3] := TRUE;   // SR flip-flop
   END_IF;
   IF #TON_TIME[6].Q THEN #"M"[3] := FALSE; END_IF;
   #TON_TIME[7].TON(IN := #"M"[3], PT := "数据块_1".到达时间);
   #Q[3] := #TON_TIME[7].Q;
END_REGION

REGION Network 6: M100.1 1口2号箱
   #_w1 := "Tag_123" AND NOT #M1[4];   // rising edge of "Tag_123"
   #M1[4] := "Tag_123";
   #TON_TIME[8].TON(IN := #Q[4], PT := "数据块_1".分拣时间);
   IF #_w1 THEN
       #"M"[4] := TRUE;   // SR flip-flop
   END_IF;
   IF #TON_TIME[8].Q THEN #"M"[4] := FALSE; END_IF;
   #TON_TIME[9].TON(IN := #"M"[4], PT := "数据块_1".到达时间);
   #Q[4] := #TON_TIME[9].Q;
END_REGION

REGION Network 7: M100.2
   #_w1 := "Tag_124" AND NOT #M1[5];   // rising edge of "Tag_124"
   #M1[5] := "Tag_124";
   #TON_TIME[10].TON(IN := #Q[5], PT := "数据块_1".分拣时间);
   IF #_w1 THEN
       #"M"[5] := TRUE;   // SR flip-flop
   END_IF;
   IF #TON_TIME[10].Q THEN #"M"[5] := FALSE; END_IF;
   #TON_TIME[11].TON(IN := #"M"[5], PT := "数据块_1".到达时间);
   #Q[5] := #TON_TIME[11].Q;
END_REGION

REGION Network 8: M100.3
   #_w1 := "Tag_125" AND NOT #M1[6];   // rising edge of "Tag_125"
   #M1[6] := "Tag_125";
   #TON_TIME[12].TON(IN := #Q[6], PT := "数据块_1".分拣时间);
   IF #_w1 THEN
       #"M"[6] := TRUE;   // SR flip-flop
   END_IF;
   IF #TON_TIME[12].Q THEN #"M"[6] := FALSE; END_IF;
   #TON_TIME[13].TON(IN := #"M"[6], PT := "数据块_1".到达时间);
   #Q[6] := #TON_TIME[13].Q;
END_REGION

REGION Network 9: M100.4
   #_w1 := "Tag_126" AND NOT #M1[7];   // rising edge of "Tag_126"
   #M1[7] := "Tag_126";
   #TON_TIME[14].TON(IN := #Q[7], PT := "数据块_1".分拣时间);
   IF #_w1 THEN
       #"M"[7] := TRUE;   // SR flip-flop
   END_IF;
   IF #TON_TIME[14].Q THEN #"M"[7] := FALSE; END_IF;
   #TON_TIME[15].TON(IN := #"M"[7], PT := "数据块_1".到达时间);
   #Q[7] := #TON_TIME[15].Q;
END_REGION

REGION Network 10 (SCL)
   REGION 4口8号
       // Statement section REGION
       IF #Q[0] OR #Q[1] OR #Q[2] OR #Q[3] THEN
           "4组正转" := TRUE;
       ELSE
           "4组正转" := FALSE;
       END_IF;
   END_REGION


   REGION 4口7号
       // Statement section REGION
       IF #Q[4] OR #Q[5] OR #Q[6] OR #Q[7] THEN
           "4组反转" := TRUE;
       ELSE
           "4组反转" := FALSE;
       END_IF;
   END_REGION
END_REGION
END_FUNCTION_BLOCK

FUNCTION_BLOCK "5口"   // FB5, LAD
{ S7_Optimized_Access := 'TRUE' }
VERSION : 0.1
   VAR_INPUT
      光电 : Bool;
      箱号 : Int;
   END_VAR
   VAR_OUTPUT
      Q : Array[0..12] of Bool;
   END_VAR
   VAR
      TON_TIME : Array[0..21] of TON_TIME;
      IEC_Timer : Array[0..11] of IEC_TIMER;
      "M" : Array[0..11] of Bool;
      M1 : Array[0..11] of Bool;
      光电上升沿 : Bool;
   END_VAR
   VAR_TEMP   // added for the SCL form of the ladder/FBD networks
      _w1 : Bool;
      _w2 : Bool;
      _w3 : Bool;
   END_VAR
BEGIN

REGION Network 1: 记录箱号
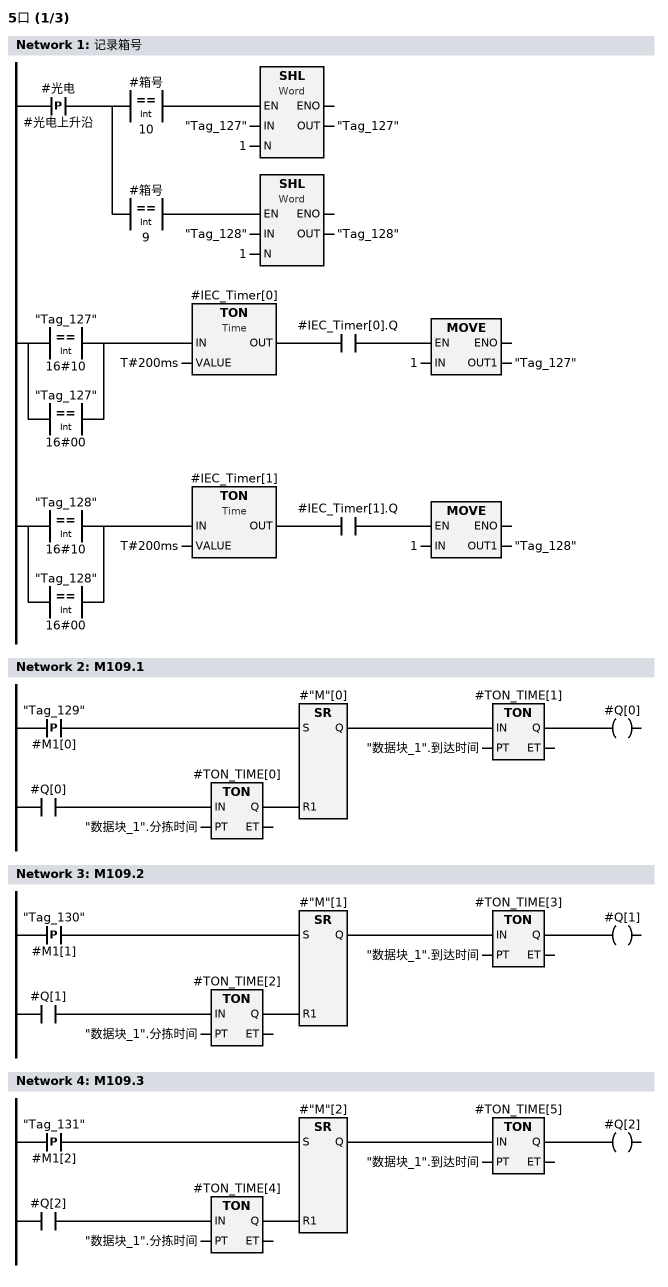
   #_w1 := #光电 AND NOT #光电上升沿;   // rising edge of #光电
   #光电上升沿 := #光电;
   IF #_w1 AND (#箱号 = 10) THEN "Tag_127" := SHL(IN := "Tag_127", N := 1); END_IF;
   IF #_w1 AND (#箱号 = 9) THEN "Tag_128" := SHL(IN := "Tag_128", N := 1); END_IF;
   #_w2 := ("Tag_127" = 16#10) OR ("Tag_127" = 16#00);
   #IEC_Timer[0].TON(IN := #_w2, PT := T#200ms);   // TON coil
   IF #_w2 AND #IEC_Timer[0].Q THEN "Tag_127" := 1; END_IF;
   #_w3 := ("Tag_128" = 16#10) OR ("Tag_128" = 16#00);
   #IEC_Timer[1].TON(IN := #_w3, PT := T#200ms);   // TON coil
   IF #_w3 AND #IEC_Timer[1].Q THEN "Tag_128" := 1; END_IF;
END_REGION

REGION Network 2: M109.1
   #_w1 := "Tag_129" AND NOT #M1[0];   // rising edge of "Tag_129"
   #M1[0] := "Tag_129";
   #TON_TIME[0].TON(IN := #Q[0], PT := "数据块_1".分拣时间);
   IF #_w1 THEN
       #"M"[0] := TRUE;   // SR flip-flop
   END_IF;
   IF #TON_TIME[0].Q THEN #"M"[0] := FALSE; END_IF;
   #TON_TIME[1].TON(IN := #"M"[0], PT := "数据块_1".到达时间);
   #Q[0] := #TON_TIME[1].Q;
END_REGION

REGION Network 3: M109.2
   #_w1 := "Tag_130" AND NOT #M1[1];   // rising edge of "Tag_130"
   #M1[1] := "Tag_130";
   #TON_TIME[2].TON(IN := #Q[1], PT := "数据块_1".分拣时间);
   IF #_w1 THEN
       #"M"[1] := TRUE;   // SR flip-flop
   END_IF;
   IF #TON_TIME[2].Q THEN #"M"[1] := FALSE; END_IF;
   #TON_TIME[3].TON(IN := #"M"[1], PT := "数据块_1".到达时间);
   #Q[1] := #TON_TIME[3].Q;
END_REGION

REGION Network 4: M109.3
   #_w1 := "Tag_131" AND NOT #M1[2];   // rising edge of "Tag_131"
   #M1[2] := "Tag_131";
   #TON_TIME[4].TON(IN := #Q[2], PT := "数据块_1".分拣时间);
   IF #_w1 THEN
       #"M"[2] := TRUE;   // SR flip-flop
   END_IF;
   IF #TON_TIME[4].Q THEN #"M"[2] := FALSE; END_IF;
   #TON_TIME[5].TON(IN := #"M"[2], PT := "数据块_1".到达时间);
   #Q[2] := #TON_TIME[5].Q;
END_REGION

REGION Network 5: M109.4
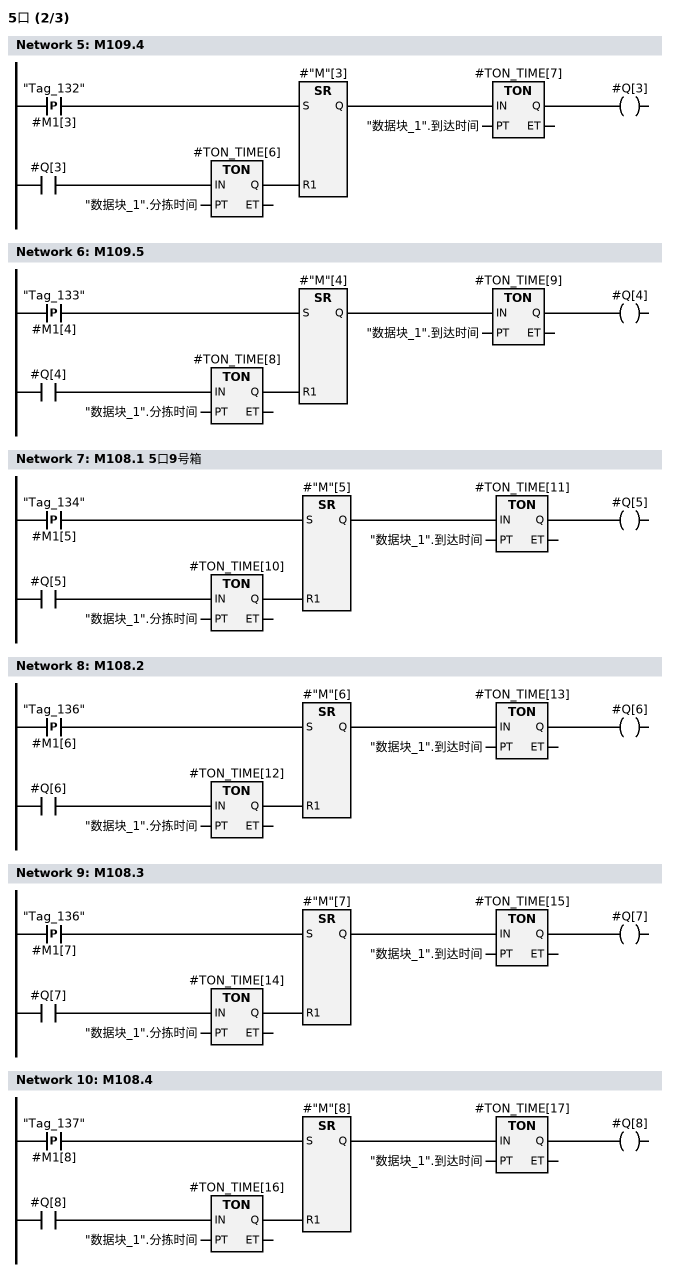
   #_w1 := "Tag_132" AND NOT #M1[3];   // rising edge of "Tag_132"
   #M1[3] := "Tag_132";
   #TON_TIME[6].TON(IN := #Q[3], PT := "数据块_1".分拣时间);
   IF #_w1 THEN
       #"M"[3] := TRUE;   // SR flip-flop
   END_IF;
   IF #TON_TIME[6].Q THEN #"M"[3] := FALSE; END_IF;
   #TON_TIME[7].TON(IN := #"M"[3], PT := "数据块_1".到达时间);
   #Q[3] := #TON_TIME[7].Q;
END_REGION

REGION Network 6: M109.5
   #_w1 := "Tag_133" AND NOT #M1[4];   // rising edge of "Tag_133"
   #M1[4] := "Tag_133";
   #TON_TIME[8].TON(IN := #Q[4], PT := "数据块_1".分拣时间);
   IF #_w1 THEN
       #"M"[4] := TRUE;   // SR flip-flop
   END_IF;
   IF #TON_TIME[8].Q THEN #"M"[4] := FALSE; END_IF;
   #TON_TIME[9].TON(IN := #"M"[4], PT := "数据块_1".到达时间);
   #Q[4] := #TON_TIME[9].Q;
END_REGION

REGION Network 7: M108.1 5口9号箱
   #_w1 := "Tag_134" AND NOT #M1[5];   // rising edge of "Tag_134"
   #M1[5] := "Tag_134";
   #TON_TIME[10].TON(IN := #Q[5], PT := "数据块_1".分拣时间);
   IF #_w1 THEN
       #"M"[5] := TRUE;   // SR flip-flop
   END_IF;
   IF #TON_TIME[10].Q THEN #"M"[5] := FALSE; END_IF;
   #TON_TIME[11].TON(IN := #"M"[5], PT := "数据块_1".到达时间);
   #Q[5] := #TON_TIME[11].Q;
END_REGION

REGION Network 8: M108.2
   #_w1 := "Tag_136" AND NOT #M1[6];   // rising edge of "Tag_136"
   #M1[6] := "Tag_136";
   #TON_TIME[12].TON(IN := #Q[6], PT := "数据块_1".分拣时间);
   IF #_w1 THEN
       #"M"[6] := TRUE;   // SR flip-flop
   END_IF;
   IF #TON_TIME[12].Q THEN #"M"[6] := FALSE; END_IF;
   #TON_TIME[13].TON(IN := #"M"[6], PT := "数据块_1".到达时间);
   #Q[6] := #TON_TIME[13].Q;
END_REGION

REGION Network 9: M108.3
   #_w1 := "Tag_136" AND NOT #M1[7];   // rising edge of "Tag_136"
   #M1[7] := "Tag_136";
   #TON_TIME[14].TON(IN := #Q[7], PT := "数据块_1".分拣时间);
   IF #_w1 THEN
       #"M"[7] := TRUE;   // SR flip-flop
   END_IF;
   IF #TON_TIME[14].Q THEN #"M"[7] := FALSE; END_IF;
   #TON_TIME[15].TON(IN := #"M"[7], PT := "数据块_1".到达时间);
   #Q[7] := #TON_TIME[15].Q;
END_REGION

REGION Network 10: M108.4
   #_w1 := "Tag_137" AND NOT #M1[8];   // rising edge of "Tag_137"
   #M1[8] := "Tag_137";
   #TON_TIME[16].TON(IN := #Q[8], PT := "数据块_1".分拣时间);
   IF #_w1 THEN
       #"M"[8] := TRUE;   // SR flip-flop
   END_IF;
   IF #TON_TIME[16].Q THEN #"M"[8] := FALSE; END_IF;
   #TON_TIME[17].TON(IN := #"M"[8], PT := "数据块_1".到达时间);
   #Q[8] := #TON_TIME[17].Q;
END_REGION

REGION Network 11: M108.5
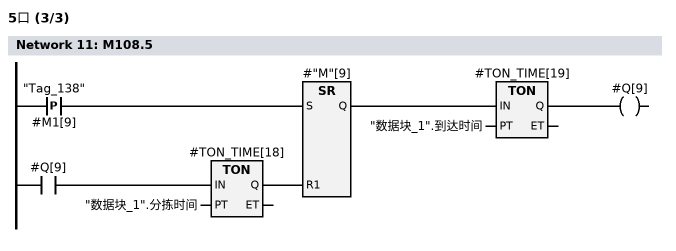
   #_w1 := "Tag_138" AND NOT #M1[9];   // rising edge of "Tag_138"
   #M1[9] := "Tag_138";
   #TON_TIME[18].TON(IN := #Q[9], PT := "数据块_1".分拣时间);
   IF #_w1 THEN
       #"M"[9] := TRUE;   // SR flip-flop
   END_IF;
   IF #TON_TIME[18].Q THEN #"M"[9] := FALSE; END_IF;
   #TON_TIME[19].TON(IN := #"M"[9], PT := "数据块_1".到达时间);
   #Q[9] := #TON_TIME[19].Q;
END_REGION

REGION Network 12 (SCL)
   REGION 5口10号
       // Statement section REGION
       IF #Q[0] OR #Q[1] OR #Q[2] OR #Q[3] OR #Q[4] THEN
           "5组正转" := TRUE;
       ELSE
           "5组正转" := FALSE;
       END_IF;
   END_REGION


   REGION 5口9号
       // Statement section REGION
       IF  #Q[5] OR #Q[6] OR #Q[7] OR #Q[8] THEN
           "5组反转" := TRUE;
       ELSE
           "5组反转" := FALSE;
       END_IF;
   END_REGION
END_REGION
END_FUNCTION_BLOCK

ORGANIZATION_BLOCK "Main"   // OB1, LAD, ProgramCycle
TITLE = "Main Program Sweep (Cycle)"
{ S7_Optimized_Access := 'TRUE' }
VERSION : 0.1
   VAR_INPUT
      Initial_Call : Bool;   // Initial call of this OB
      Remanence : Bool;   // =True, if remanent data are available
   END_VAR
BEGIN

REGION Network 1
   // 变频器运行
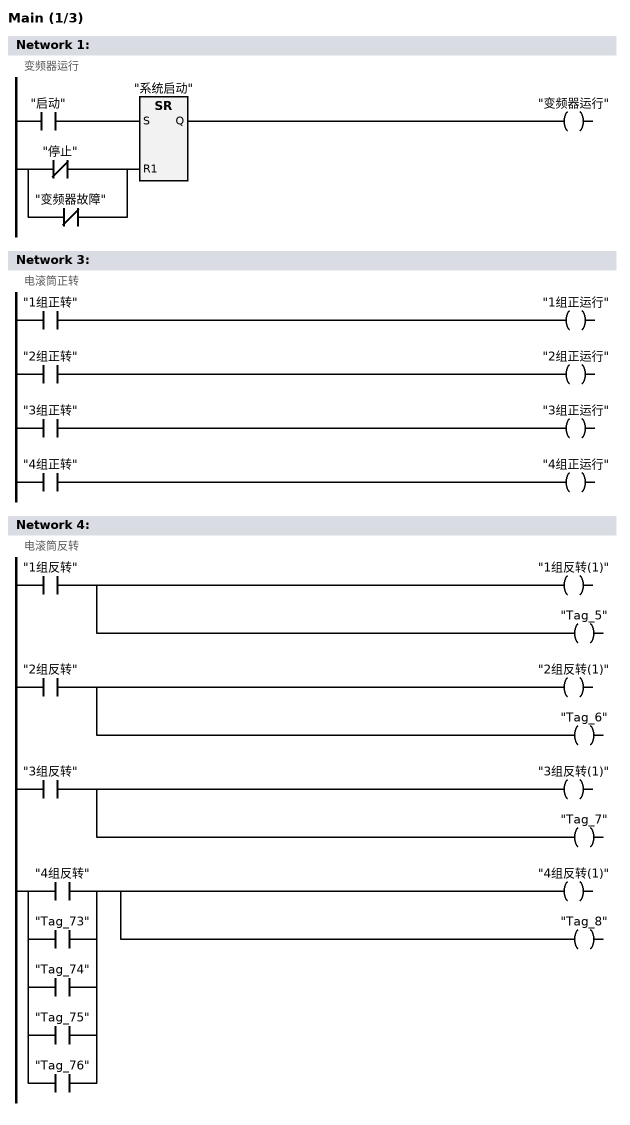
   RUNG wire#powerrail
      Contact( "启动" )
      S_SR(operand := "系统启动", r1 := wire#w1)
      Coil( "变频器运行" )
   END_RUNG
   RUNG wire#powerrail
      I_Contact( "停止" )
   END_RUNG wire#w1
   RUNG wire#powerrail
      I_Contact( "变频器故障" )
   END_RUNG wire#w1
   // the same network as SCL:
   IF "启动" THEN
       "系统启动" := TRUE;   // SR flip-flop
   END_IF;
   IF NOT "停止" OR NOT "变频器故障" THEN "系统启动" := FALSE; END_IF;
   "变频器运行" := "系统启动";
END_REGION

REGION Network 3
   // 电滚筒正转
   RUNG wire#powerrail
      Contact( "1组正转" )
      Coil( "1组正运行" )
   END_RUNG
   RUNG wire#powerrail
      Contact( "2组正转" )
      Coil( "2组正运行" )
   END_RUNG
   RUNG wire#powerrail
      Contact( "3组正转" )
      Coil( "3组正运行" )
   END_RUNG
   RUNG wire#powerrail
      Contact( "4组正转" )
      Coil( "4组正运行" )
   END_RUNG
   // the same network as SCL:
   "1组正运行" := "1组正转";
   "2组正运行" := "2组正转";
   "3组正运行" := "3组正转";
   "4组正运行" := "4组正转";
END_REGION

REGION Network 4
   // 电滚筒反转
   RUNG wire#powerrail
      Contact( "1组反转" )
      wire#w1
      Coil( "1组反转(1)" )
   END_RUNG
   RUNG wire#w1
      Coil( "Tag_5" )
   END_RUNG
   RUNG wire#powerrail
      Contact( "2组反转" )
      wire#w2
      Coil( "2组反转(1)" )
   END_RUNG
   RUNG wire#w2
      Coil( "Tag_6" )
   END_RUNG
   RUNG wire#powerrail
      Contact( "3组反转" )
      wire#w3
      Coil( "3组反转(1)" )
   END_RUNG
   RUNG wire#w3
      Coil( "Tag_7" )
   END_RUNG
   RUNG wire#powerrail
      Contact( "4组反转" )
      wire#w4
      Coil( "4组反转(1)" )
   END_RUNG
   RUNG wire#powerrail
      Contact( "Tag_73" )
   END_RUNG wire#w4
   RUNG wire#powerrail
      Contact( "Tag_74" )
   END_RUNG wire#w4
   RUNG wire#powerrail
      Contact( "Tag_75" )
   END_RUNG wire#w4
   RUNG wire#powerrail
      Contact( "Tag_76" )
   END_RUNG wire#w4
   RUNG wire#w4
      Coil( "Tag_8" )
   END_RUNG
   // the same network as SCL:
   "1组反转(1)" := "1组反转";
   "Tag_5" := "1组反转";
   "2组反转(1)" := "2组反转";
   "Tag_6" := "2组反转";
   "3组反转(1)" := "3组反转";
   "Tag_7" := "3组反转";
   "4组反转(1)" := "4组反转" OR "Tag_73" OR "Tag_74" OR "Tag_75" OR "Tag_76";
   "Tag_8" := "4组反转(1)";
END_REGION

REGION Network 5
   // 三基色绿色
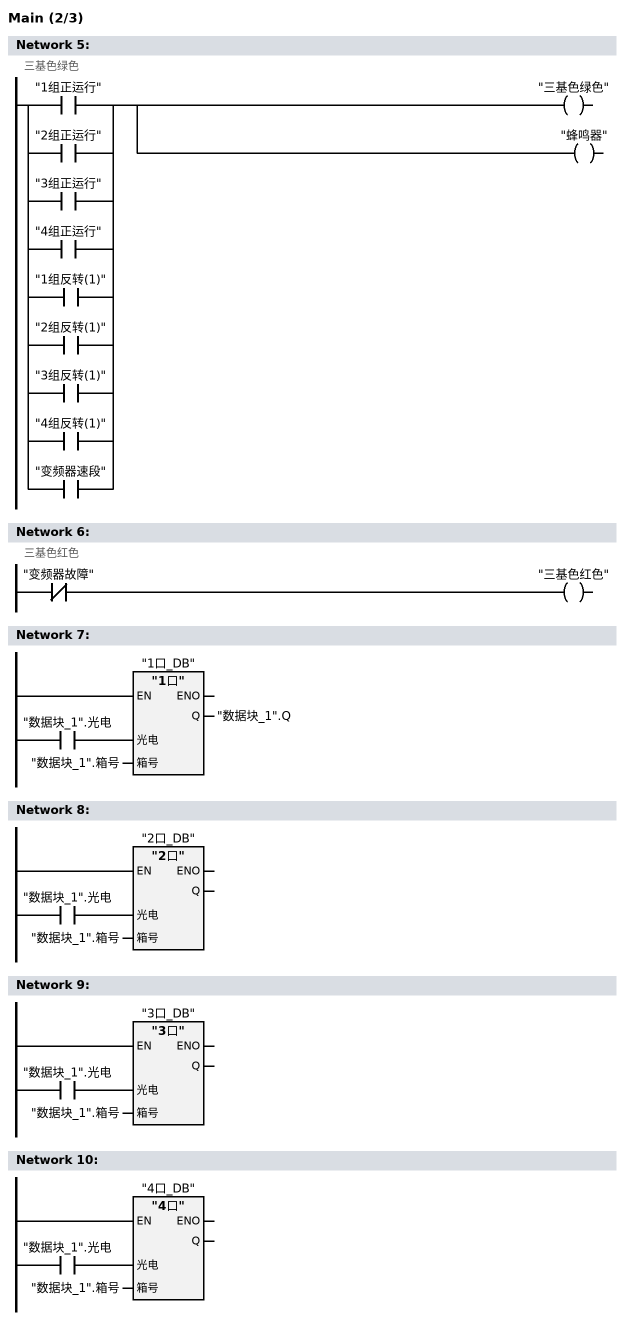
   RUNG wire#powerrail
      Contact( "1组正运行" )
      wire#w1
      Coil( "三基色绿色" )
   END_RUNG
   RUNG wire#powerrail
      Contact( "2组正运行" )
   END_RUNG wire#w1
   RUNG wire#powerrail
      Contact( "3组正运行" )
   END_RUNG wire#w1
   RUNG wire#powerrail
      Contact( "4组正运行" )
   END_RUNG wire#w1
   RUNG wire#powerrail
      Contact( "1组反转(1)" )
   END_RUNG wire#w1
   RUNG wire#powerrail
      Contact( "2组反转(1)" )
   END_RUNG wire#w1
   RUNG wire#powerrail
      Contact( "3组反转(1)" )
   END_RUNG wire#w1
   RUNG wire#powerrail
      Contact( "4组反转(1)" )
   END_RUNG wire#w1
   RUNG wire#powerrail
      Contact( "变频器速段" )
   END_RUNG wire#w1
   RUNG wire#w1
      Coil( "蜂鸣器" )
   END_RUNG
   // the same network as SCL:
   "三基色绿色" := "1组正运行" OR "2组正运行" OR "3组正运行" OR "4组正运行" OR "1组反转(1)" OR "2组反转(1)" OR "3组反转(1)" OR "4组反转(1)" OR "变频器速段";
   "蜂鸣器" := "三基色绿色";
END_REGION

REGION Network 6
   // 三基色红色
   RUNG wire#powerrail
      I_Contact( "变频器故障" )
      Coil( "三基色红色" )
   END_RUNG
   // the same network as SCL:
   "三基色红色" := NOT "变频器故障";
END_REGION

REGION Network 7
   RUNG wire#powerrail
      "1口_DB"(光电 := wire#w1, 箱号 := "数据块_1".箱号, Q => "数据块_1".Q)
   END_RUNG
   RUNG wire#powerrail
      Contact( "数据块_1".光电 )
   END_RUNG wire#w1
   // the same network as SCL:
   "1口_DB"(光电 := "数据块_1".光电, 箱号 := "数据块_1".箱号, Q => "数据块_1".Q);   // "1口"
END_REGION

REGION Network 8
   RUNG wire#powerrail
      "2口_DB"(光电 := wire#w1, 箱号 := "数据块_1".箱号, Q =>)
   END_RUNG
   RUNG wire#powerrail
      Contact( "数据块_1".光电 )
   END_RUNG wire#w1
   // the same network as SCL:
   "2口_DB"(光电 := "数据块_1".光电, 箱号 := "数据块_1".箱号);   // "2口"
END_REGION

REGION Network 9
   RUNG wire#powerrail
      "3口_DB"(光电 := wire#w1, 箱号 := "数据块_1".箱号, Q =>)
   END_RUNG
   RUNG wire#powerrail
      Contact( "数据块_1".光电 )
   END_RUNG wire#w1
   // the same network as SCL:
   "3口_DB"(光电 := "数据块_1".光电, 箱号 := "数据块_1".箱号);   // "3口"
END_REGION

REGION Network 10
   RUNG wire#powerrail
      "4口_DB"(光电 := wire#w1, 箱号 := "数据块_1".箱号, Q =>)
   END_RUNG
   RUNG wire#powerrail
      Contact( "数据块_1".光电 )
   END_RUNG wire#w1
   // the same network as SCL:
   "4口_DB"(光电 := "数据块_1".光电, 箱号 := "数据块_1".箱号);   // "4口"
END_REGION

REGION Network 11
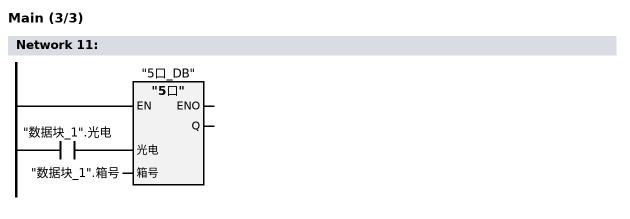
   RUNG wire#powerrail
      "5口_DB"(光电 := wire#w1, 箱号 := "数据块_1".箱号, Q =>)
   END_RUNG
   RUNG wire#powerrail
      Contact( "数据块_1".光电 )
   END_RUNG wire#w1
   // the same network as SCL:
   "5口_DB"(光电 := "数据块_1".光电, 箱号 := "数据块_1".箱号);   // "5口"
END_REGION
END_ORGANIZATION_BLOCK